FUNCTION alg_g_a_X2: REAL
{ S7_Optimized_Access := 'false' }
    VAR_INPUT
        state: STATE;
    END_VAR

BEGIN
    alg_g_a_X2 := state.curTime;
END_FUNCTION
